FUNCTION_BLOCK TRAJECTORY_VIEWER_COMM (* Sends geom_file *)
  (* Standard: 61499-2 *)
  (* Version 1.0, 03-07-12, GASR, Universidade do Estado de Santa Catarina *)
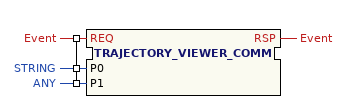
  EVENT_INPUT
    REQ WITH P0, P1; (* Request file storage *)
  END_EVENT
  EVENT_OUTPUT
    RSP; (* Finished operation *)
  END_EVENT
  VAR_INPUT
    P0 : STRING := COEF_FILE; (* Filename *)
    P1 : ANY; (* Var1 *)
  END_VAR
END_FUNCTION_BLOCK
